// Basic passive digital-input CM. Owning logic consumes semantic Value; the
// project catalog injects the physical identity separately from the HAL.
FUNCTION_BLOCK FB_DigitalInputCM EXTENDS FB_ControlModuleBase
VAR_INPUT
    ParCfg : ST_DigitalInputParCfg;
    ParCmd : ST_DigitalInputParCmd;
END_VAR
VAR_OUTPUT
    OutCmd : ST_DigitalInputOutCmd;
    OutImm : ST_DigitalInputOutImm;
END_VAR
VAR
    {attribute 'OPC.UA.DA' := '0'}
    _hal : REFERENCE TO ST_DigitalInputHal;
    _identity : ST_IoPointIdentity;
END_VAR

Cyclic();

METHOD Setup : BOOL
VAR_INPUT
    Name : STRING(80);
    HalRef : REFERENCE TO ST_DigitalInputHal;
    DisplayNameKey : STRING(160);
    DescriptionKey : STRING(160);
END_VAR
_M_SetName(Name);
_M_SetPresentation(DisplayNameKey := DisplayNameKey, DescriptionKey := DescriptionKey, TypeKey := 'std.moduleType.digitalInput');
_hal REF= HalRef;
Setup := __ISVALIDREF(_hal);
END_METHOD

METHOD ConfigureIoIdentity
VAR_INPUT
    Identity : ST_IoPointIdentity;
END_VAR
_identity := Identity;
END_METHOD

METHOD PROTECTED OnCyclic : DINT
OnCyclic := SUPER^.OnCyclic();
IF __ISVALIDREF(_hal) THEN
    OutImm.Value := _hal.Value;
    OutImm.Quality := _hal.Quality;
ELSE
    OutImm.Value := FALSE;
    OutImm.Quality := FALSE;
END_IF
OutImm.IoTag := _identity.Tag;
OutImm.Diagnostic := Status.Diagnostic;
END_METHOD

METHOD PROTECTED _M_Dispatch
_M_Fault(E_Reason.UNSUPPORTED_COMMAND,
    'std.error.passiveInputHasNoCommand');
END_METHOD

METHOD PROTECTED _M_PublishStatus
SUPER^._M_PublishStatus();
OutImm.Diagnostic := Status.Diagnostic;
END_METHOD

END_FUNCTION_BLOCK

(* stored: Version 1.1.0.1, ProductVersion 3.1.4024.12
   POU FB_DigitalInputCM: Id {bef0d2f4-c055-483d-87bd-71220916a9c8}, SpecialFunc None
   Method Setup: Id {b70106bd-7c20-4eb4-9f60-84b9b573029d}
   Method ConfigureIoIdentity: Id {789228a1-b030-462d-87c0-971c9df0b9b1}
   Method OnCyclic: Id {db657fb3-2810-452c-9365-29a71eab4373}
   Method _M_Dispatch: Id {e15aca44-e2b0-4382-a45f-cbbefbe8d5a2}
   Method _M_PublishStatus: Id {ec384437-4c0b-4098-b960-6f8ef7a4915b} *)
